Universal Robots PolyScope program: matlabcoontrol3dmouse.urp

ProgramRoot setBeforeStartSequence=true; directory=/programs/usbdisk/UR5RobotControlV3.1/UR5RobotControlV3/PolyScope; kinematics=(a=[0, -0.425, -0.39225, 0, 0, 0], d=[0.08916, 0, 0, 0.10915, 0.09465, 0.0823], alpha=[1.5708, 0, 0, 1.5708, -1.5708, 0], deltaTheta=[0, 0, 0, 0, 0, 0], status=notInitialized); name=matlabcoontrol3dmouse; programVersion=(project__name=PolyScope, major__version=1, minor__version=8, svn__revision=11657, build__date=Oct 09 2013, 20:14:19); robotEnvironmentFileName=default; serialNumberRobot=2013215294
  BeforeStart description=COMMAND_SEQUENCE_BEFORE_PROGRAM_START; name=BeforeStart
    Assignment assignmentValueSource=0; expr=[6,0,0,0,0,0,0]; operatorValueType=INTEGER; valueSource=EXPRESSION; variable=(name=receive_data, prefersPersistentValue=false, requestANewUniqueName=false)
    Assignment assignmentValueSource=0; expr=[0,0,0,0,0,0]; operatorValueType=INTEGER; valueSource=EXPRESSION; variable=(name=Move_To_Pos, prefersPersistentValue=false, requestANewUniqueName=false)
    Script type=0; expressionBranchNode=pose_1=get_forward_kin()
    Assignment assignmentValueSource=0; expr=0; operatorValueType=INTEGER; valueSource=EXPRESSION; variable=(name=pointer, prefersPersistentValue=false, requestANewUniqueName=false)
    While count=0; expr=ExpressionVariableNode<ExpressionVariableNode[0]; type=LOOP_EXPR; variable=(name=Loop_2, prefersPersistentValue=false, requestANewUniqueName=false)
      Script type=0; expressionBranchNode=Move_To_Pos[pointer]=pose_1[pointer]
      Assignment assignmentValueSource=0; expr=ExpressionVariableNode+1; operatorValueType=INTEGER; valueSource=EXPRESSION; variable=(name=pointer, prefersPersistentValue=false, requestANewUniqueName=false)
    Script type=0; expressionBranchNode=socket_open("192.168.73.1",30000)
    Assignment assignmentValueSource=0; expr=[0,0]; operatorValueType=INTEGER; valueSource=EXPRESSION; variable=(name=task, prefersPersistentValue=false, requestANewUniqueName=false)
    Assignment assignmentValueSource=0; expr=[0,0,0,0,0,0]; operatorValueType=INTEGER; valueSource=EXPRESSION; variable=(name=Move_To_Pos, prefersPersistentValue=false, requestANewUniqueName=false)
  MainProgram cartesianAcceleration=1.2; cartesianSpeed=0.25; jointAcceleration=1.3962634015954636; jointSpeed=1.0471975511965976; moveAsFastAsPossible=true; sharedProcessMoveBlendRadius=0.025; motionType=JOINT_SPACE; variableFeature=___tran51ate_this_name___Joint_0_name
    Script type=0; expressionBranchNode=ExpressionVariableNode=socket_read_ascii_float(1)
    If expr=ExpressionVariableNode[1]≟1; type=IF_NODE
      CallSubProgram subProgramNodeToCall=receive_data=socket_read_ascii_float(6)
      Assignment assignmentValueSource=0; expr=[0,0]; operatorValueType=INTEGER; valueSource=EXPRESSION; variable=(name=task, prefersPersistentValue=false, requestANewUniqueName=false)
    If expr=ExpressionVariableNode[1]≟2; type=ELSEIF_NODE
      CallSubProgram subProgramNodeToCall=pose_1=get_forward_kin()
      Assignment assignmentValueSource=0; expr=[0,0]; operatorValueType=INTEGER; valueSource=EXPRESSION; variable=(name=task, prefersPersistentValue=false, requestANewUniqueName=false)
    Wait analogComparison=0; analogInputRange=0; analogValue=0.0; digitalValue=0; selectedAnalogSensor=-1; selectedDigitalSensor=-1; waitTime=0.01; type=TIMER_WAIT
  Thread name=Thread_1
    Script type=0; expressionBranchNode=speedl(Move_To_Pos,a=0.5,t_min=0.01)
  subProgramToCall name=SubProgram_1
    Script type=0; expressionBranchNode=receive_data=socket_read_ascii_float(6)
    If expr=ExpressionVariableNode[0]≠6; type=IF_NODE
      Script type=0; expressionBranchNode=socket_send_string("0")
    If type=ELSE_NODE
      Script type=0; expressionBranchNode=socket_send_string("1")
      Assignment assignmentValueSource=0; expr=0; operatorValueType=INTEGER; valueSource=EXPRESSION; variable=(name=pointer, prefersPersistentValue=false, requestANewUniqueName=false)
      While count=0; expr=ExpressionVariableNode<ExpressionVariableNode[0]; type=LOOP_EXPR; variable=(name=Loop_1, prefersPersistentValue=false, requestANewUniqueName=false)
        Script type=0; expressionBranchNode=Move_To_Pos[pointer]=receive_data[pointer+1]
        Assignment assignmentValueSource=0; expr=ExpressionVariableNode+1; operatorValueType=INTEGER; valueSource=EXPRESSION; variable=(name=pointer, prefersPersistentValue=false, requestANewUniqueName=false)
  subProgramToCall name=SubProgram_2
    Script type=0; expressionBranchNode=pose_1=get_forward_kin()
    Script type=0; expressionBranchNode=socket_send_string(pose_1)
